{attribute addProperty BoxType "EL9930-0000-0016"}
{attribute addProperty Id "A_0002_EL9930_0001_0016EL9930_AECBF7E8324A_0003_EL9930_0000_0017A_0003_EL9930_0000_0017_B9BF5D41324"}
{attribute addProperty CRC "3209054368"}
{attribute addProperty SizeInBites "64"}
{attribute addProperty SizeInBytes "8"}
TYPE A_0001_EL9930_0000_0016_BF4648A0 EXTENDS EL9930_E441AFC3 :
STRUCT
	{attribute addProperty Name "A_0002_EL9930_0001_0016"}
	A_0002_EL9930_0001_0016 : EL9930_AECBF7E8;
	{attribute addProperty Name "A_0003_EL9930_0000_0017"}
	A_0003_EL9930_0000_0017 : A_0003_EL9930_0000_0017_B9BF5D41;
END_STRUCT
END_TYPE

(* stored: Version 1.2.0.0, ProductVersion 3.1.4024.9
   DUT A_0001_EL9930_0000_0016_BF4648A0: Id {1f7bb6a7-1e86-4188-9182-4a8d70da1568} *)
